//FUNCTION_BLOCK TcAxis_Tc3_DriveMotionControl EXTENDS TcAxis_Base IMPLEMENTS itfAxis_Tc3_DriveMotionControl
//FUNCTION_BLOCK TcAxis_Tc3_DriveMotionControl EXTENDS TcAxis_Base
FUNCTION_BLOCK TcAxis_Tc3_DriveMotionControl IMPLEMENTS itfAxis_Tc3_DriveMotionControl
//VAR_INPUT
//END_VAR
//VAR_OUTPUT
//END_VAR
VAR_IN_OUT 
	Axis 				: Tc3_DriveMotionControl.AXIS_REF();
END_VAR
VAR
	_PowerOn 			: BOOL;
	_fbAxisCommand   	: TcAxisCommand;
	MC 					: ST_Tc3_DriveMotionControl;
END_VAR

{warning 'Agregar implementación de método'}
METHOD AbortTrigger : itfCommand
END_METHOD

{warning 'Agregar implementación de propiedad'}
PROPERTY ActualPosition : REAL
GET
END_GET
END_PROPERTY

{warning 'Agregar implementación de propiedad'}
PROPERTY ActualVelocity : REAL
GET
END_GET
END_PROPERTY

{warning 'Agregar implementación de propiedad'}
PROPERTY Error : BOOL
GET
END_GET
END_PROPERTY

{warning 'Agregar implementación de propiedad'}
PROPERTY ErrorId : WORD
GET
END_GET
END_PROPERTY

{warning 'Agregar implementación de propiedad'}
PROPERTY ErrorId_Udint_Status : UDINT
GET
END_GET
END_PROPERTY

{attribute 'TcRpcEnable'}
METHOD Halt : itfAxisCommand
VAR_INPUT
	Deceleration	: REAL;
	Jerk	: REAL;
	BufferMode	: MC_BUFFER_MODE;
END_VAR
END_METHOD

{attribute 'TcRpcEnable'}
METHOD Home : itfAxisCommand
VAR_INPUT
	Position	: REAL;
	Velocity	: REAL;
	EndVelocity	: REAL;
	Acceleration	: REAL;
	Deceleration	: REAL;
	Jerk	: REAL;
	Direction	: MC_Direction;
	HomingMode	: INT;
	BufferMode	: MC_BUFFER_MODE;
END_VAR
END_METHOD

{warning 'Agregar implementación de propiedad'}
PROPERTY IsHomed : BOOL
GET
END_GET
END_PROPERTY

{attribute 'TcRpcEnable'}
METHOD Jog : itfAxisCommand
VAR_INPUT
	JogForward	: BOOL;
	JogBackwards	: BOOL;
	Mode	: Tc2_MC2.E_JogMode;
	Position	: LREAL;
	Velocity	: LREAL;
	Acceleration	: LREAL;
	Deceleration	: LREAL;
	Jerk	: LREAL;
END_VAR
END_METHOD

{warning 'Agregar implementación de propiedad'}
PROPERTY MotionStatus : MOTION_STATUS
GET
END_GET
END_PROPERTY

{attribute 'TcRpcEnable'}
METHOD MoveAbsolute : itfAxisCommand
VAR_INPUT
	Position		: REAL;
	Velocity		: REAL;
	Acceleration	: REAL;
	Deceleration	: REAL;
	Jerk			: REAL;
//	Direction		: MC_Direction;
	BufferMode		: MC_BUFFER_MODE;
//	Options         : Tc2_MC2.ST_MoveOptions;
	Options         : ST_MoveOptions;
END_VAR

VAR
	itfAxisCommand   : itfAxisCommand;
    _Command         : ST_Command;
END_VAR
itfAxisCommand := _fbAxisCommand;
	
MC.MoveAbsolute(
	Axis:= Axis, 
	Execute:= TRUE ,
	Position:= Position, 
	Velocity:= Velocity, 
	Acceleration:= Acceleration, 
	Deceleration:= Deceleration, 
	Options:= ,//,Options, 
	Done=> _Command.Done, 
	Busy=> _Command.Busy, 
	Active=>_Command.Active, 
	CommandAborted=> _Command.CommandAborted, 
	Error=> _Command.Error, 
	ErrorID=> _Command.ErrorID_Udint);
	
MC.MoveAbsolute(
	Axis:= Axis, 
	Execute:= FALSE);	

itfAxisCommand.Done 				:=  _Command.Done AND ActualPosition = Position;             
itfAxisCommand.Busy   				:=	_Command.Busy;
itfAxisCommand.Active 				:=	_Command.Active;
itfAxisCommand.CommandAborted		:=	_Command.CommandAborted;
itfAxisCommand.Error 				:=	_Command.Error;
itfAxisCommand.ErrorID_Udint 		:=	_Command.ErrorID_Udint;

MoveAbsolute := itfAxisCommand;
END_METHOD

{attribute 'TcRpcEnable'}
METHOD MoveModulo : itfAxisCommand
END_METHOD

{attribute 'TcRpcEnable'}
METHOD MoveRelative : itfAxisCommand
VAR_INPUT
	Distance	: REAL;
	Velocity	: REAL;
	Acceleration	: REAL;
	Deceleration	: REAL;
	Jerk	: REAL;
	BufferMode	: MC_BUFFER_MODE;
END_VAR
END_METHOD

{attribute 'TcRpcEnable'}
METHOD MoveVelocity : itfContinuousAxisCommand
VAR_INPUT
	Velocity	: REAL;
	Acceleration	: REAL;
	Deceleration	: REAL;
	Jerk	: REAL;
	Direction	: MC_Direction;
	BufferMode	: MC_BUFFER_MODE;
END_VAR
END_METHOD

{attribute 'TcRpcEnable'}
METHOD Power : itfCommand
VAR_INPUT
	Enable	: BOOL;
	EnablePositive	: BOOL;
	EnableNegative	: BOOL;
END_VAR
VAR
	_fbCommand      : TcCommand;
	itfCommand      : itfCommand;
	Command         : ST_Command;
END_VAR

itfCommand := _fbCommand;

MC.Power(
	Axis:= Axis, 
	Enable:= Enable, 
	Status=> Command.Status, 
	Busy=> Command.Busy, 
	Active=> Command.Active, 
	Error=> Command.Error, 
	ErrorID=> Command.ErrorID_Udint);
	
itfCommand.Status		:=	Command.Status;
itfCommand.Busy   		:=	Command.Busy;
itfCommand.Active 		:=	Command.Active;
itfCommand.Error 		:=	Command.Error;
itfCommand.ErrorID_Udint :=	Command.ErrorID_Udint;
	
Power := itfCommand;

_PowerOn := MC.Power.Enable;
END_METHOD

{warning 'Agregar implementación de propiedad'}
PROPERTY PowerOn : BOOL
GET
END_GET
END_PROPERTY

{attribute 'TcRpcEnable'}
METHOD Reset : itfCommand
END_METHOD

{attribute 'TcRpcEnable'}
METHOD SetPosition : itfCommand
VAR_INPUT
	Position	: REAL;
	Relative	: BOOL;
	(*	ExecutionMode	: MC_ExecutionMode;*)
	ExecutionMode	: Tc2_MC2.ST_SetPositionOptions;
END_VAR
END_METHOD

{warning 'Agregar implementación de propiedad'}
PROPERTY Simulation : BOOL
GET
END_GET
END_PROPERTY

{warning 'Agregar implementación de propiedad'}
PROPERTY Status : MC_AxisStates
GET
VAR
	AxisStates : MC_AxisStates;
END_VAR
CASE Axis.Status.MotionState OF 
    MC_AXISSTATE_UNDEFINED : 
         AxisStates := MC_AxisStates.MC_AXISSTATE_UNDEFINED;
	MC_AXISSTATE_DISABLED:
		AxisStates := MC_AxisStates.MC_AXISSTATE_DISABLED;
	MC_AXISSTATE_STANDSTILL:
		AxisStates := MC_AxisStates.MC_AXISSTATE_STANDSTILL;
	MC_AXISSTATE_ERRORSTOP:		
		AxisStates := MC_AxisStates.MC_AXISSTATE_ERRORSTOP;
	MC_AXISSTATE_STOPPING:			
		AxisStates := MC_AxisStates.MC_AXISSTATE_STOPPING;
	MC_AXISSTATE_HOMING:			
		AxisStates := MC_AxisStates.MC_AXISSTATE_HOMING;
	MC_AXISSTATE_DISCRETEMOTION:			
		AxisStates := MC_AxisStates.MC_AXISSTATE_DISCRETEMOTION;
	MC_AXISSTATE_CONTINOUSMOTION:			
		AxisStates := MC_AxisStates.MC_AXISSTATE_CONTINOUSMOTION;
//	MC_AXISSTATE_SYNCHRONIZEDMOTION:			
//		AxisStates := MC_AxisStates.MC_AXISSTATE_SYNCHRONIZEDMOTION;
END_CASE;

Status := AxisStates;
END_GET
END_PROPERTY

{attribute 'TcRpcEnable'}
METHOD Stop : itfAxisCommand
VAR_INPUT
	Deceleration	: REAL;
	Jerk	: REAL;
END_VAR
END_METHOD

{warning 'Agregar implementación de método'}
METHOD TouchProbe : itfCommand
END_METHOD

END_FUNCTION_BLOCK

(* stored: Version 1.1.0.1, ProductVersion 3.1.4024.12
   POU TcAxis_Tc3_DriveMotionControl: Id {3ecf364f-113f-4c6b-b875-0e5527cca083}, SpecialFunc None
   Folder ActualValues: Id {464c5fc7-15fd-4283-9600-38274052a8b4}
   Folder Control: Id {6cdffade-85fb-4f5d-8a7c-c71bb3170518}
   Folder SingleAxisMotion: Id {b7925eff-99b2-4831-a464-5f49b517660c}
   Folder Status: Id {6645e220-d671-4ff7-9366-a23923b75211}
   Folder Touch Probe: Id {0e54e46b-72b5-4574-99fb-da3e9944f20d}
   Method AbortTrigger: Id {feab4aa0-5203-4852-94a9-c32cc42b9d39}
   Property ActualPosition: Id {e30305a4-d564-4e3f-ad84-9b2c24b49032}
   Get Get: Id {3220cda9-a83a-47c0-8f33-9712834bf809}
   Property ActualVelocity: Id {b963a623-d580-4903-9ba5-a1264f89b0f6}
   Get Get: Id {ebe076c4-8acf-4da1-bd0a-d7f7d6141baf}
   Property Error: Id {1b2d3d6a-4c39-49c2-9f8c-12da2391e304}
   Get Get: Id {e2b09937-aea1-46ab-b504-246be2554405}
   Property ErrorId: Id {803e65e4-594c-4dd5-a441-b694c0587443}
   Get Get: Id {2157a368-a75a-4a90-bf22-af491bd7499c}
   Property ErrorId_Udint_Status: Id {ad6b1f80-d466-4ce5-b2f3-77e0d35b29f3}
   Get Get: Id {7d230420-8954-4074-8722-b665db6cf3a0}
   Method Halt: Id {955fbd7d-c030-408d-afe3-691e208b6d21}
   Method Home: Id {295f9667-97ab-4fef-8431-c56488c0ce43}
   Property IsHomed: Id {993f97cb-ea6a-45fc-a1dd-08a75c2b28f8}
   Get Get: Id {00bb9c5c-e890-4eab-b759-4eafa83eaf7f}
   Method Jog: Id {623021d8-2cdb-46ff-acbd-868a96d59581}
   Property MotionStatus: Id {22de4599-0e89-4380-99e8-d701c9ca0327}
   Get Get: Id {880a167c-c982-4a1f-8ea8-e280dc3d2630}
   Method MoveAbsolute: Id {83d876d4-3b03-4f0f-9a15-b15c1a9a76bd}
   Method MoveModulo: Id {1a34a205-a66a-489a-ac35-79ff51afa913}
   Method MoveRelative: Id {892d2412-1304-44be-a52e-798f5976d6af}
   Method MoveVelocity: Id {51c35689-c199-4411-8e3a-a8b21bff495b}
   Method Power: Id {94b47b09-3379-4705-94af-80b852c42c93}
   Property PowerOn: Id {91f5fe00-793f-465e-b14b-8962261961e3}
   Get Get: Id {d2555f19-3709-4ccf-a489-5b925040bc8f}
   Method Reset: Id {3fc0ed87-e795-46d0-b18a-a6fd89904168}
   Method SetPosition: Id {2b189c3e-5b6f-429f-963f-350a39320a4b}
   Property Simulation: Id {e5bbd793-62e5-41e0-bd62-f66f1bb77738}
   Get Get: Id {2195b2a2-03d0-436f-a463-f49389ba3c10}
   Property Status: Id {a7f35970-5385-4014-972b-e1c724acbf81}
   Get Get: Id {595291b0-7d83-45e8-84c6-c1638d4ab754}
   Method Stop: Id {2d28494d-9637-4f56-b05f-8de95af50c48}
   Method TouchProbe: Id {74a3236d-eacb-42fe-a95e-6e303ed17b1a} *)
